PROGRAM MAIN
VAR
	nState,i: INT;
	fbR_TrigExecute : R_Trig;
	StartSafety :BOOL := TRUE;
	
	TcRestart : TC_Restart;
	Restart : BOOL;
	busy : BOOL;
	State AT%I* :ARRAY[1..2] OF UINT;
END_VAR

FOR i := 1 TO 8 DO 
	GVL_io.Voltage[i]:= SQRT( EXP(GVL_io.D_Spannung[i]) + EXP(GVL_io.Q_Spannung[i]));
END_FOR


IF GVL_Safety.hwStart THEN
	StartSafety := TRUE;
	GVL_Safety.Run := TRUE;
	GVL_Safety.Start := TRUE;

ELSIF NOT GVL_Safety.hwStop	THEN 
	StartSafety := FALSE;
END_IF

GVL_Safety.Reset := GVL_Safety.hwReset  OR Restart;

 GVL_Safety.HW_Error :=  State[1] <> 8 OR  State[2] <> 8  ;
GVL_Safety.HW_Ok  :=GVL_Safety.SaeftyOk;

 GVL_Safety.HW_Reset_Req:= (GVL_Safety.Error_Other OR GVL_Safety.Error_Out OR GVL_Safety.Error_Com );
(*
TcRestart(
	NETID:= '', 
	RESTART:=Restart , 
	TMOUT:= , 
	BUSY=> busy, 
	ERR=> , 
	ERRID=> );
	
	*)

METHOD Safety : BOOL

VAR_INPUT
	bExecute : BOOL;
END_VAR

VAR

END_VAR
fbR_TrigExecute(CLK := bExecute);
IF fbR_TrigExecute.Q   THEN
	nState := 10;		
ELSIF NOT bExecute THEN
	nState := 0;
	GVL_Safety.Run := FALSE;
	
END_IF

CASE nState OF
	 0: // Wait State
	 	
	10: 
		GVL_Safety.Run := TRUE;
		GVL_Safety.Start := TRUE;
		GVL_Safety.Reset := TRUE;
		nState :=20;
	15:

		GVL_Safety.Reset := FALSE;
		nState :=200;

			
	20:
		GVL_Safety.Reset := FALSE;

		IF 	GVL_Safety.SaeftyOk THEN
			nState :=99;
			Safety := TRUE;
		ELSIF 	(GVL_Safety.Error_Other OR GVL_Safety.Error_Out OR GVL_Safety.Error_Com )  THEN 
		
			nState :=15;
		END_IF
	40:
		GVL_Safety.reset := TRUE;
		IF NOT (GVL_Safety.Error_Other OR GVL_Safety.Error_Out OR GVL_Safety.Error_Com )THEN
			GVL_Safety.Reset := FALSE;
			nState :=99;
		END_IF	
	99: 
		IF NOT GVL_Safety.SaeftyOk THEN
			nState :=40;
			Safety := TRUE;
		END_IF

	
END_CASE
END_METHOD

END_PROGRAM

(* stored: Version 1.1.0.1, ProductVersion 3.1.4024.12
   POU MAIN: Id {1b4dff48-5fc4-4640-872d-67c650f13b5e}, SpecialFunc None
   Method Safety: Id {5e78818f-12cb-483c-81e6-defbcc3ed4ae} *)
